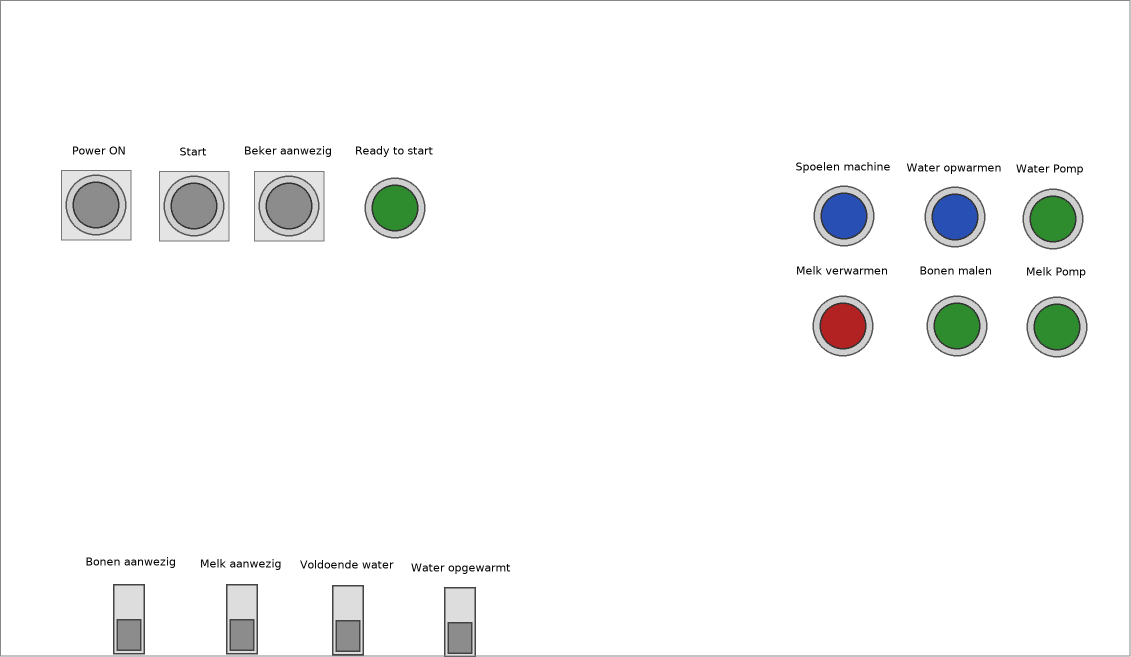
VISUALIZATION Visualization  // 1131x657
    Lamp1 (809,181 70x70), tooltip "Spoelen machine", variable: GVL.Spoelen_machine, style: Lamp-Lamp1-Blue
    PushSwitch (61,170 70x70), variable: GVL.Power_ON, behaviour: TOGGLE, style: Switch-PushSwitch-Gray
    Label (768,152 150x30), "Spoelen machine"
    Lamp1 (360,173 70x70), variable: Proces_1.Led_ready_start, style: Lamp-Lamp1-Green
    Label (319,136 150x30), "Ready to start"
    DipSwitch (94,584 70x70), variable: Proces_1.Bonen_aanwezig, behaviour: TOGGLE, style: Switch-DipSwitch-Gray
    Label (56,547 150x30), "Bonen aanwezig"
    Label (166,549 150x30), "Melk aanwezig"
    DipSwitch (207,584 70x70), variable: Proces_1.Melk_aanwezig, behaviour: TOGGLE, style: Switch-DipSwitch-Gray
    Label (272,550 150x30), "Voldoende water"
    DipSwitch (313,585 70x70), variable: Proces_1.Voldoende_water, behaviour: TOGGLE, style: Switch-DipSwitch-Gray
    Lamp1 (920,182 70x70), variable: GVL.Water_verwarmen, style: Lamp-Lamp1-Blue
    Label (879,153 150x30), "Water opwarmen"
    DipSwitch (425,587 70x70), variable: GVL.Water_opgewarmt, behaviour: TOGGLE, style: Switch-DipSwitch-Gray
    Label (386,553 150x30), "Water opgewarmt"
    Label (24,136 150x30), "Power ON"
    PushSwitch (159,171 70x70), variable: Proces_1.Start, behaviour: TOGGLE, style: Switch-PushSwitch-Gray
    Label (118,137 150x30), "Start"
    PushSwitch (254,171 70x70), variable: Proces_1.Beker_aanwezig, behaviour: TOGGLE, style: Switch-PushSwitch-Gray
    Label (213,136 150x30), "Beker aanwezig"
    Lamp1 (808,291 70x70), variable: Proces_1.Melk_verwarming, style: Lamp-Lamp1-Red
    Label (767,256 150x30), "Melk verwarmen"
    Label (981,257 150x30), "Melk Pomp"
    Lamp1 (1022,292 70x70), variable: Proces_1.Melk_pomp, style: Lamp-Lamp1-Green
    Label (881,256 150x30), "Bonen malen"
    Lamp1 (922,291 70x70), variable: Proces_1.Bonen_malen, style: Lamp-Lamp1-Green
    Lamp1 (1018,184 70x70), variable: Proces_1.Water_pomp, style: Lamp-Lamp1-Green
    Label (975,154 150x30), "Water Pomp"
END_VISUALIZATION

(* stored: Version 1.1.0.1, ProductVersion 3.1.4024.12
   Visu Visualization: Id {b18016b9-03d7-4df7-be4f-e0407d37d4bb} *)
